FUNCTION_BLOCK FB_TestSuite2 EXTENDS FB_TestSuite
VAR_INPUT
END_VAR
VAR_OUTPUT
END_VAR
VAR
END_VAR

TestCase2A();
TestCase2B();

TEST('TestCase2C');

AssertTrue(TRUE, 'Condition is not true');
AssertTrue(FALSE, 'Condition is not true');

TEST_FINISHED();

METHOD PUBLIC Method_CFC : BOOL
VAR_INPUT
END_VAR
END_METHOD

METHOD PUBLIC Method_FBD : BOOL
VAR_INPUT
END_VAR
// NETWORK 1
END_METHOD

METHOD PUBLIC Method_LD : BOOL
VAR_INPUT
END_VAR
// NETWORK 1
END_METHOD

METHOD PUBLIC Method_UML : REFERENCE TO FB_Test
VAR_INPUT
END_VAR
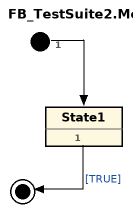
STATECHART Method_UML  // abortable
    START StartState1
    STATE State1
    END EndState1
    StartState1 -> State1  // priority 1, on completion
    State1 -> EndState1 [TRUE] // priority 1
END_STATECHART
END_METHOD

METHOD TestCase2A
VAR_INPUT
END_VAR
TEST('TestCase2A');

AssertTrue(TRUE, 'Condition is not true');

TEST_FINISHED();
END_METHOD

METHOD TestCase2B
VAR_INPUT
END_VAR
TEST('TestCase2B');

AssertTrue(TRUE, 'Condition is not true');
AssertTrue(TRUE, 'Condition is not true');

TEST_FINISHED();
END_METHOD

END_FUNCTION_BLOCK

(* stored: Version 1.1.0.1, ProductVersion 3.1.4024.12
   POU FB_TestSuite2: Id {3a6274d6-6083-4f38-89f5-174a468b61d8}, SpecialFunc None
   Method Method_CFC: Id {6220ef8c-b93c-4d03-82f1-d0fb0e0f8f17}
   Method Method_FBD: Id {89216776-ec63-4446-89c7-6f879b632364}
   Method Method_LD: Id {ed18b6ba-a455-4ed5-ba73-d77ee2c19325}
   Method Method_UML: Id {75329e18-c2b7-42f7-9e4e-69f84cf1fe42}
   Method TestCase2A: Id {08302e5c-315f-491e-adf5-28ac987840cc}
   Method TestCase2B: Id {d124f6c2-5ec2-4271-8a1e-818da4d1bf79} *)
